Staubli VAL3: main.pgx

public program main()
begin
  // INIT
  call onStart()
  // LOOP UNTIL nKey=255
  do
    call refresh()
    nKey=getKey()
    call use:listevent(nKey,nFrame,sEvent)
    nView=use:nView
    switch nKey
      case 259
        // TAB
        bLarge=!bLarge
        call use:setView(bLarge)
      break
      case 263
        call onBackEvent()
      break
      case 271
        call onF1Event()
      break
      case 272
        call onF2Event()
      break
      case 273
        call onF3Event()
      break
      case 274
        call onF4Event()
      break
      case 275
        call onF5Event()
      break
      case 276
        call onF6Event()
      break
      case 277
        call onF7Event()
      break
      case 278
        call onF8Event()
      break
      case 270
        call onEnterEvent()
      break
    endSwitch
    // release the resource
    delay(0)
  until nKey==255
  // on Exit
  call onExit()
end
